PROGRAM Tips_and_tricks
VAR
END_VAR

// Shortcuts

// Comment muliple lines of code: CTRL + K, CTRL + U
// Uncomment multiple lines of code : CTRL + K, CTRL + U

END_PROGRAM

(* stored: Version 1.1.0.1, ProductVersion 3.1.4024.13
   POU Tips_and_tricks: Id {8f2bc4d2-f867-495c-a56d-85046e3b6546}, SpecialFunc None *)
